FUNCTION_BLOCK FB_Animal
VAR
	 sOutput : STRING := '';
	 
	  x : INT := 8;
END_VAR

METHOD M_Eat
VAR_INPUT
END_VAR
THIS^.sOutput := 'Animal eats food';
END_METHOD

METHOD M_Sleep : BOOL
VAR_INPUT
END_VAR
THIS^.sOutput := 'Animal sleeps';
END_METHOD

END_FUNCTION_BLOCK

(* stored: Version 1.1.0.1, ProductVersion 3.1.4024.16
   POU FB_Animal: Id {8daf69df-8f2e-49d0-8756-076b96a34518}, SpecialFunc None
   Method M_Eat: Id {1649086b-5256-41da-aee6-0fbc9699b7fe}
   Method M_Sleep: Id {cc7a2d05-88b8-44dc-801c-c6d84e1e38c7} *)
